(* IEC 61131-3 sources: neuroplc/results/scl_output (part 2) *)

      // MatMul 'l0_base': W + bias
      w2[0] := 0.6531532; w2[1] := 1.1509302; w2[2] := 0.8542801; w2[3] := 0.1212990; w2[4] := 0.6904182; w2[5] := -0.5414373; w2[6] := -0.9088417; w2[7] := -0.5722627;
      w2[8] := 0.8944874; w2[9] := 0.5538955; w2[10] := -1.0278374; w2[11] := -0.4903141; w2[12] := -0.1389806; w2[13] := 0.4674363; w2[14] := -1.0210936; w2[15] := -0.6274210;
      w2[16] := 0.2741612; w2[17] := 1.0625501; w2[18] := -0.9149109; w2[19] := -0.7328060; w2[20] := 0.7575151; w2[21] := -0.2042419; w2[22] := -0.2723309; w2[23] := -0.7191657;
      w2[24] := -0.0280776; w2[25] := 0.2011455; w2[26] := -0.3273573; w2[27] := -0.4418836; w2[28] := 1.2626092; w2[29] := 1.2265757; w2[30] := 1.5492810; w2[31] := -0.5662438;
      w2[32] := -0.9511591; w2[33] := 0.1725382; w2[34] := 1.2004387; w2[35] := -0.0104933; w2[36] := 1.5757133; w2[37] := 1.6623878; w2[38] := 1.2453479; w2[39] := 0.1729178;
      w2[40] := 0.2919613; w2[41] := 0.0309749; w2[42] := -0.6492561; w2[43] := -0.3796145; w2[44] := -0.5120577; w2[45] := 0.3172240; w2[46] := -0.4038502; w2[47] := 0.5928957;
      w2[48] := -0.5418487; w2[49] := -0.5144768; w2[50] := -0.7627655; w2[51] := 0.8234128; w2[52] := -0.4605753; w2[53] := -0.7895154; w2[54] := 0.0910844; w2[55] := -0.6752480;
      w2[56] := 0.0697802; w2[57] := -0.4284368; w2[58] := 0.0479970; w2[59] := 0.0784096; w2[60] := -0.0238369; w2[61] := 0.0168181; w2[62] := -0.8319796; w2[63] := 0.1763645;
      w2[64] := 0.2104895; w2[65] := 0.8926834; w2[66] := 0.6908084; w2[67] := 0.4001502; w2[68] := -0.3938401; w2[69] := 0.1085153; w2[70] := -0.6449838; w2[71] := -0.7566856;
      w2[72] := -0.0827282; w2[73] := 0.4948159; w2[74] := -1.1559126; w2[75] := -0.5277553; w2[76] := 0.8248507; w2[77] := 0.1181727; w2[78] := 0.7966241; w2[79] := 0.2058670;
      w2[80] := -0.8326430; w2[81] := -0.1626337; w2[82] := -0.0323979; w2[83] := -0.2344580; w2[84] := -1.5619131; w2[85] := -1.4697499; w2[86] := -1.8048265; w2[87] := -0.8762984;
      w2[88] := -1.3497895; w2[89] := -0.8686097; w2[90] := -0.9026392; w2[91] := -0.7284883; w2[92] := -1.7362306; w2[93] := -0.0363061; w2[94] := 1.1192808; w2[95] := 0.8043320;
      w2[96] := -0.1950512; w2[97] := -0.3716736; w2[98] := -0.4853409; w2[99] := -0.5649784; w2[100] := -0.4172391; w2[101] := 0.6161152; w2[102] := -0.6759697; w2[103] := 0.0904574;
      w2[104] := 0.5806844; w2[105] := 0.6348718; w2[106] := 0.7333751; w2[107] := 0.6839716; w2[108] := -0.3869329; w2[109] := 0.5344537; w2[110] := 0.9650685; w2[111] := 0.0383124;
      w2[112] := -0.8913731; w2[113] := -0.3576556; w2[114] := -0.6536014; w2[115] := -0.0847967; w2[116] := -0.0349820; w2[117] := 0.5889089; w2[118] := -0.2677067; w2[119] := -0.2245978;
      w2[120] := -0.5749647; w2[121] := -0.9168990; w2[122] := -0.6333076; w2[123] := -0.4074411; w2[124] := 0.4441338; w2[125] := 0.1501607; w2[126] := -0.1995225; w2[127] := 0.7596117;
      w2[128] := 0.0808029; w2[129] := -0.3484810; w2[130] := -0.0210259; w2[131] := 0.9137757; w2[132] := -0.7801852; w2[133] := -0.2238004; w2[134] := -0.3275166; w2[135] := -0.0392269;
      w2[136] := -0.2500529; w2[137] := 0.1511434; w2[138] := -0.2167200; w2[139] := 0.2951781; w2[140] := 0.3186197; w2[141] := 0.0769461; w2[142] := 0.4348049; w2[143] := -0.2419707;
      w2[144] := -0.3043656; w2[145] := -0.3270995; w2[146] := 0.5164679; w2[147] := 0.4538959; w2[148] := 0.2316195; w2[149] := 0.8929619; w2[150] := 1.3953813; w2[151] := 0.6482492;
      w2[152] := -0.2139386; w2[153] := -0.0555586; w2[154] := -0.2996079; w2[155] := -0.7336348; w2[156] := -0.7894226; w2[157] := 0.6769296; w2[158] := -1.0865229; w2[159] := 0.9084685;
      w2[160] := 0.4970312; w2[161] := 0.3730805; w2[162] := 0.6737831; w2[163] := 0.5160832; w2[164] := -0.8191277; w2[165] := 0.0919100; w2[166] := 0.4878978; w2[167] := -0.4577431;
      w2[168] := 0.5415249; w2[169] := 0.0459770; w2[170] := 0.2380498; w2[171] := 0.3544105; w2[172] := 0.0758338; w2[173] := 0.5700713; w2[174] := -0.3280728; w2[175] := 0.0073880;
      w2[176] := 0.9576581; w2[177] := -0.1927161; w2[178] := -0.5408630; w2[179] := 0.3759742; w2[180] := -0.3697540; w2[181] := -0.4095958; w2[182] := 0.2953050; w2[183] := -0.3224963;
      w2[184] := 0.4659955; w2[185] := 0.2666524; w2[186] := 0.7817978; w2[187] := -0.3882965; w2[188] := 0.5259117; w2[189] := 0.1157550; w2[190] := -0.0868794; w2[191] := 0.1442592;
      w2[192] := 0.4463586; w2[193] := -0.0788809; w2[194] := 0.3359323; w2[195] := 0.3131578; w2[196] := -0.2152938; w2[197] := 0.8472598; w2[198] := 0.6115276; w2[199] := -0.3911876;
      w2[200] := 0.0704370; w2[201] := -0.2515413; w2[202] := 0.8549601; w2[203] := 0.3596184; w2[204] := -0.5991781; w2[205] := -1.2437032; w2[206] := -0.1800027; w2[207] := -1.1388100;
      w2[208] := 0.5647227; w2[209] := 0.3254773; w2[210] := -0.8980638; w2[211] := 0.6457720; w2[212] := 0.9825901; w2[213] := -0.7528893; w2[214] := 0.0748151; w2[215] := 0.1365464;
      w2[216] := -0.6619212; w2[217] := -0.1892451; w2[218] := -0.3664528; w2[219] := -0.7725444; w2[220] := -0.1610090; w2[221] := -0.1782233; w2[222] := -0.1539104; w2[223] := -0.0613308;
      w2[224] := 1.0186411; w2[225] := -0.0857887; w2[226] := -0.3516517; w2[227] := 0.3065239; w2[228] := 0.0238268; w2[229] := 0.2399618; w2[230] := -0.2922754; w2[231] := -0.1875871;
      w2[232] := 1.1885412; w2[233] := -0.1608811; w2[234] := -1.1761448; w2[235] := -0.3997688; w2[236] := -1.0060421; w2[237] := 0.0516912; w2[238] := 0.4627137; w2[239] := -1.1369811;
      w2[240] := 0.6643242; w2[241] := 0.2780860; w2[242] := 0.0209994; w2[243] := -0.6893836; w2[244] := 0.5776726; w2[245] := -0.0303992; w2[246] := -0.2795104; w2[247] := -0.2218146;
      w2[248] := 0.4949092; w2[249] := 0.1933563; w2[250] := -0.3510525; w2[251] := 0.0224845; w2[252] := -1.5212339; w2[253] := -1.1815313; w2[254] := -1.4145346; w2[255] := 0.4340951;
      w2[256] := 0.3062091; w2[257] := 0.0455918; w2[258] := -0.3191082; w2[259] := 0.2872083; w2[260] := -1.7960831; w2[261] := -0.9681343; w2[262] := -0.2131347; w2[263] := -0.0914112;
      w2[264] := 0.4054331; w2[265] := -0.9982103; w2[266] := -0.5022178; w2[267] := 0.3359171; w2[268] := 0.8721167; w2[269] := -0.0940284; w2[270] := -1.9242376; w2[271] := 0.1256431;
      w2[272] := -0.4745836; w2[273] := 0.5358467; w2[274] := 0.1780284; w2[275] := -0.2262570; w2[276] := -0.6270480; w2[277] := -0.4930463; w2[278] := -0.6283804; w2[279] := 0.2633540;
      w2[280] := 0.2300479; w2[281] := 1.1844879; w2[282] := 0.6107946; w2[283] := -0.2428536; w2[284] := 0.4828842; w2[285] := 0.1695227; w2[286] := 0.5681323; w2[287] := 0.2884444;
      w2[288] := 0.2841129; w2[289] := -0.8758434; w2[290] := 0.2491129; w2[291] := -0.3859273; w2[292] := -0.4150312; w2[293] := 0.4644483; w2[294] := 0.1481924; w2[295] := -0.4265237;
      w2[296] := 0.3190451; w2[297] := -0.6888376; w2[298] := 0.8258311; w2[299] := 0.4234703; w2[300] := 0.0811714; w2[301] := -0.2619098; w2[302] := -1.0289083; w2[303] := -0.8263102;
      w2[304] := 0.5947338; w2[305] := -0.0104262; w2[306] := 0.4936709; w2[307] := 0.0368680; w2[308] := 0.0356015; w2[309] := 0.8885249; w2[310] := 0.5964210; w2[311] := -0.0492413;
      w2[312] := -0.1171272; w2[313] := -0.2020979; w2[314] := 0.5844330; w2[315] := -0.0603527; w2[316] := -0.1831383; w2[317] := -1.3109881; w2[318] := -0.5292199; w2[319] := 0.0204109;
      w2[320] := 0.2865884; w2[321] := -0.0319725; w2[322] := -0.1081036; w2[323] := 0.6079996; w2[324] := 0.7452201; w2[325] := -0.9360539; w2[326] := 0.2803982; w2[327] := 0.5940919;
      w2[328] := -0.3924443; w2[329] := -0.0010045; w2[330] := -0.2540028; w2[331] := -0.1956804; w2[332] := 0.3307257; w2[333] := -0.0851964; w2[334] := 0.0121359; w2[335] := 0.2464700;
      w2[336] := -1.3067886; w2[337] := -1.2725198; w2[338] := -1.4913075; w2[339] := 0.6236749; w2[340] := 0.3114894; w2[341] := 0.3706363; w2[342] := -0.5315891; w2[343] := 0.3905119;
      w2[344] := -1.4648223; w2[345] := -0.4327554; w2[346] := -0.1879684; w2[347] := -0.2010098; w2[348] := 0.5315167; w2[349] := -0.0843144; w2[350] := 0.0634309; w2[351] := 0.3992346;
      w2[352] := 0.3824810; w2[353] := -0.0483803; w2[354] := -0.2913157; w2[355] := 0.0982564; w2[356] := -0.4671767; w2[357] := 0.1136492; w2[358] := 0.0548117; w2[359] := -0.2728889;
      w2[360] := -0.4076180; w2[361] := -0.4225101; w2[362] := -0.2261286; w2[363] := 0.2782121; w2[364] := 0.7695327; w2[365] := 0.2566034; w2[366] := 0.1953621; w2[367] := 0.0408440;
      w2[368] := 0.0124786; w2[369] := 0.2488524; w2[370] := -0.5697264; w2[371] := 0.0825308; w2[372] := 0.8317476; w2[373] := -0.8402474; w2[374] := -1.0685767; w2[375] := -0.2165811;
      w2[376] := -0.4149429; w2[377] := -0.3753743; w2[378] := 0.1834853; w2[379] := 0.0865243; w2[380] := 0.7913322; w2[381] := -0.3387795; w2[382] := 0.5137359; w2[383] := -0.3165046;
      w2[384] := 0.2458227; w2[385] := 0.3609711; w2[386] := -0.3399727; w2[387] := -0.8827292; w2[388] := 0.4816631; w2[389] := 0.3397982; w2[390] := 0.1536530; w2[391] := 0.1695612;
      w2[392] := 0.5854009; w2[393] := -0.0813269; w2[394] := 0.1311246; w2[395] := 0.0674454; w2[396] := 0.2877986; w2[397] := -0.2290608; w2[398] := -0.6208226; w2[399] := -0.5486314;
      w2[400] := 0.9404889; w2[401] := 0.4580346; w2[402] := -0.5092251; w2[403] := -0.5765274; w2[404] := -0.4888373; w2[405] := 0.0444687; w2[406] := -0.2916232; w2[407] := -0.8206158;
      w2[408] := 0.2447187; w2[409] := 0.4721361; w2[410] := -0.6585346; w2[411] := -0.6879834; w2[412] := 0.5628800; w2[413] := 0.0532022; w2[414] := 0.1965619; w2[415] := 0.0561261;
      w2[416] := 0.2354458; w2[417] := 0.3610592; w2[418] := 0.0144084; w2[419] := 0.1184748; w2[420] := 0.0501975; w2[421] := 0.1787246; w2[422] := 0.4878071; w2[423] := 0.1703812;
      w2[424] := 0.1714815; w2[425] := -0.0600145; w2[426] := 0.7518312; w2[427] := 0.4750999; w2[428] := -0.1374112; w2[429] := 1.2641517; w2[430] := 1.2422327; w2[431] := 0.3578296;
      w2[432] := -0.3659381; w2[433] := 0.3438349; w2[434] := -0.3962274; w2[435] := -0.3011864; w2[436] := -0.1204108; w2[437] := 0.3932763; w2[438] := -0.0552154; w2[439] := 0.3200105;
      w2[440] := 0.7434683; w2[441] := 0.4552981; w2[442] := 0.4342712; w2[443] := 0.2647173; w2[444] := -0.2187249; w2[445] := -0.2678579; w2[446] := 0.1962206; w2[447] := -0.4789418;
      b3[0] := 0.0; b3[1] := 0.0; b3[2] := 0.0; b3[3] := 0.0; b3[4] := 0.0; b3[5] := 0.0; b3[6] := 0.0; b3[7] := 0.0;
      b3[8] := 0.0; b3[9] := 0.0; b3[10] := 0.0; b3[11] := 0.0; b3[12] := 0.0; b3[13] := 0.0; b3[14] := 0.0; b3[15] := 0.0;

      // BsplineLUT 'l1_bspline': grid + table
      g4[0] := -3.0000000; g4[1] := -2.5714286; g4[2] := -2.1428571; g4[3] := -1.7142857; g4[4] := -1.2857143; g4[5] := -0.8571429; g4[6] := -0.4285714; g4[7] := 0.0;
      g4[8] := 0.4285714; g4[9] := 0.8571429; g4[10] := 1.2857143; g4[11] := 1.7142857; g4[12] := 2.1428571; g4[13] := 2.5714286; g4[14] := 3.0000000;
      t5[0] := 0.1180185; t5[1] := 0.1203233; t5[2] := 0.1224589; t5[3] := 0.1244152; t5[4] := 0.1261825; t5[5] := 0.1277508; t5[6] := 0.1291103; t5[7] := 0.1302511;
      t5[8] := 0.1311632; t5[9] := 0.1318369; t5[10] := 0.1322627; t5[11] := 0.1324407; t5[12] := 0.1323814; t5[13] := 0.1320955; t5[14] := 0.1315938; t5[15] := 0.0842773;
      t5[16] := 0.0825064; t5[17] := 0.0806832; t5[18] := 0.0787976; t5[19] := 0.0768397; t5[20] := 0.0747991; t5[21] := 0.0726658; t5[22] := 0.0704296; t5[23] := 0.0680806;
      t5[24] := 0.0656084; t5[25] := 0.0630035; t5[26] := 0.0602665; t5[27] := 0.0574086; t5[28] := 0.0544416; t5[29] := 0.0513772; t5[30] := 0.0936770; t5[31] := 0.0899939;
      t5[32] := 0.0863021; t5[33] := 0.0826108; t5[34] := 0.0789293; t5[35] := 0.0752668; t5[36] := 0.0716325; t5[37] := 0.0680359; t5[38] := 0.0644860; t5[39] := 0.0609922;
      t5[40] := 0.0575636; t5[41] := 0.0542039; t5[42] := 0.0509117; t5[43] := 0.0476852; t5[44] := 0.0445227; t5[45] := 0.0226024; t5[46] := 0.0203358; t5[47] := 0.0180222;
      t5[48] := 0.0156702; t5[49] := 0.0132885; t5[50] := 0.0108859; t5[51] := 0.0084710; t5[52] := 0.0060526; t5[53] := 0.0036394; t5[54] := 0.0012401; t5[55] := -0.0011365;
      t5[56] := -0.0034818; t5[57] := -0.0057870; t5[58] := -0.0080435; t5[59] := -0.0102426; t5[60] := -0.0585543; t5[61] := -0.0502811; t5[62] := -0.0417866; t5[63] := -0.0330670;
      t5[64] := -0.0241186; t5[65] := -0.0149379; t5[66] := -0.0055211; t5[67] := 0.0041354; t5[68] := 0.0140353; t5[69] := 0.0241822; t5[70] := 0.0345793; t5[71] := 0.0452160;
      t5[72] := 0.0560676; t5[73] := 0.0671089; t5[74] := 0.0783146; t5[75] := 0.0506554; t5[76] := 0.0470260; t5[77] := 0.0433342; t5[78] := 0.0395754; t5[79] := 0.0357449;
      t5[80] := 0.0318381; t5[81] := 0.0278503; t5[82] := 0.0237768; t5[83] := 0.0196131; t5[84] := 0.0153543; t5[85] := 0.0109963; t5[86] := 0.0065434; t5[87] := 0.0020089;
      t5[88] := -0.0025934; t5[89] := -0.0072500; t5[90] := 0.0495298; t5[91] := 0.0382326; t5[92] := 0.0269749; t5[93] := 0.0157830; t5[94] := 0.0046829; t5[95] := -0.0062993;
      t5[96] := -0.0171372; t5[97] := -0.0278048; t5[98] := -0.0382758; t5[99] := -0.0485243; t5[100] := -0.0585243; t5[101] := -0.0682607; t5[102] := -0.0777291; t5[103] := -0.0869256;
      t5[104] := -0.0958461; t5[105] := 0.0110217; t5[106] := 0.0143777; t5[107] := 0.0176291; t5[108] := 0.0207730; t5[109] := 0.0238068; t5[110] := 0.0267275; t5[111] := 0.0295325;
      t5[112] := 0.0322190; t5[113] := 0.0347841; t5[114] := 0.0372252; t5[115] := 0.0395394; t5[116] := 0.0417255; t5[117] := 0.0437835; t5[118] := 0.0457136; t5[119] := 0.0475160;
      t5[120] := 0.1000672; t5[121] := 0.0975504; t5[122] := 0.0949741; t5[123] := 0.0923415; t5[124] := 0.0896557; t5[125] := 0.0869198; t5[126] := 0.0841368; t5[127] := 0.0813098;
      t5[128] := 0.0784420; t5[129] := 0.0755364; t5[130] := 0.0725962; t5[131] := 0.0696262; t5[132] := 0.0666327; t5[133] := 0.0636224; t5[134] := 0.0606016; t5[135] := -0.0637436;
      t5[136] := -0.0601492; t5[137] := -0.0563668; t5[138] := -0.0523824; t5[139] := -0.0481823; t5[140] := -0.0437526; t5[141] := -0.0390796; t5[142] := -0.0341494; t5[143] := -0.0289481;
      t5[144] := -0.0234621; t5[145] := -0.0176780; t5[146] := -0.0115977; t5[147] := -0.0052384; t5[148] := 0.0013820; t5[149] := 0.0082455; t5[150] := 0.0125032; t5[151] := 0.0077389;
      t5[152] := 0.0030834; t5[153] := -0.0014561; t5[154] := -0.0058727; t5[155] := -0.0101594; t5[156] := -0.0143091; t5[157] := -0.0183148; t5[158] := -0.0221695; t5[159] := -0.0258661;
      t5[160] := -0.0293979; t5[161] := -0.0327624; t5[162] := -0.0359621; t5[163] := -0.0389996; t5[164] := -0.0418773; t5[165] := 0.1193166; t5[166] := 0.1212150; t5[167] := 0.1228393;
      t5[168] := 0.1241749; t5[169] := 0.1252072; t5[170] := 0.1259215; t5[171] := 0.1263033; t5[172] := 0.1263380; t5[173] := 0.1260110; t5[174] := 0.1253076; t5[175] := 0.1242140;
      t5[176] := 0.1227300; t5[177] := 0.1208703; t5[178] := 0.1186500; t5[179] := 0.1160843; t5[180] := -0.1185704; t5[181] := -0.1148212; t5[182] := -0.1108735; t5[183] := -0.1067269;
      t5[184] := -0.1023809; t5[185] := -0.0978348; t5[186] := -0.0930883; t5[187] := -0.0881406; t5[188] := -0.0829914; t5[189] := -0.0776400; t5[190] := -0.0720863; t5[191] := -0.0663355;
      t5[192] := -0.0603990; t5[193] := -0.0542886; t5[194] := -0.0480157; t5[195] := 0.0583250; t5[196] := 0.0564782; t5[197] := 0.0548263; t5[198] := 0.0533813; t5[199] := 0.0521553;
      t5[200] := 0.0511605; t5[201] := 0.0504090; t5[202] := 0.0499130; t5[203] := 0.0496845; t5[204] := 0.0497356; t5[205] := 0.0500779; t5[206] := 0.0507077; t5[207] := 0.0516058;
      t5[208] := 0.0527522; t5[209] := 0.0541270; t5[210] := 0.1353638; t5[211] := 0.1313381; t5[212] := 0.1272324; t5[213] := 0.1230490; t5[214] := 0.1187897; t5[215] := 0.1144566;
      t5[216] := 0.1100518; t5[217] := 0.1055772; t5[218] := 0.1010349; t5[219] := 0.0964268; t5[220] := 0.0917550; t5[221] := 0.0870218; t5[222] := 0.0822297; t5[223] := 0.0773811;
      t5[224] := 0.0724786; t5[225] := -0.0180711; t5[226] := -0.0229253; t5[227] := -0.0277300; t5[228] := -0.0324813; t5[229] := -0.0371753; t5[230] := -0.0418079; t5[231] := -0.0463752;
      t5[232] := -0.0508733; t5[233] := -0.0552981; t5[234] := -0.0596458; t5[235] := -0.0639125; t5[236] := -0.0680959; t5[237] := -0.0721960; t5[238] := -0.0762126; t5[239] := -0.0801455;
      t5[240] := 0.1276658; t5[241] := 0.1281422; t5[242] := 0.1286489; t5[243] := 0.1291845; t5[244] := 0.1297478; t5[245] := 0.1303374; t5[246] := 0.1309519; t5[247] := 0.1315901;
      t5[248] := 0.1322506; t5[249] := 0.1329321; t5[250] := 0.1336332; t5[251] := 0.1343503; t5[252] := 0.1350780; t5[253] := 0.1358105; t5[254] := 0.1365422; t5[255] := 0.1341147;
      t5[256] := 0.1308563; t5[257] := 0.1273050; t5[258] := 0.1234552; t5[259] := 0.1193012; t5[260] := 0.1148372; t5[261] := 0.1100576; t5[262] := 0.1049567; t5[263] := 0.0995287;
      t5[264] := 0.0937679; t5[265] := 0.0876691; t5[266] := 0.0812383; t5[267] := 0.0744930; t5[268] := 0.0674512; t5[269] := 0.0601309; t5[270] := 0.0900934; t5[271] := 0.0884138;
      t5[272] := 0.0867445; t5[273] := 0.0850886; t5[274] := 0.0834493; t5[275] := 0.0818300; t5[276] := 0.0802338; t5[277] := 0.0786640; t5[278] := 0.0771239; t5[279] := 0.0756166;
      t5[280] := 0.0741453; t5[281] := 0.0727099; t5[282] := 0.0713072; t5[283] := 0.0699338; t5[284] := 0.0685862; t5[285] := 0.0413872; t5[286] := 0.0350636; t5[287] := 0.0287237;
      t5[288] := 0.0223717; t5[289] := 0.0160115; t5[290] := 0.0096474; t5[291] := 0.0032833; t5[292] := -0.0030765; t5[293] := -0.0094280; t5[294] := -0.0157671; t5[295] := -0.0220896;
      t5[296] := -0.0283901; t5[297] := -0.0346618; t5[298] := -0.0408980; t5[299] := -0.0470918; t5[300] := 0.0755875; t5[301] := 0.0739173; t5[302] := 0.0718717; t5[303] := 0.0694406;
      t5[304] := 0.0666140; t5[305] := 0.0633818; t5[306] := 0.0597340; t5[307] := 0.0556606; t5[308] := 0.0511514; t5[309] := 0.0461965; t5[310] := 0.0407865; t5[311] := 0.0349304;
      t5[312] := 0.0286561; t5[313] := 0.0219922; t5[314] := 0.0149673; t5[315] := 0.1297014; t5[316] := 0.1303879; t5[317] := 0.1309192; t5[318] := 0.1312868; t5[319] := 0.1314823;
      t5[320] := 0.1314970; t5[321] := 0.1313227; t5[322] := 0.1309508; t5[323] := 0.1303729; t5[324] := 0.1295806; t5[325] := 0.1285656; t5[326] := 0.1273265; t5[327] := 0.1258690;
      t5[328] := 0.1241989; t5[329] := 0.1223223; t5[330] := -0.0027479; t5[331] := 0.0012134; t5[332] := 0.0050790; t5[333] := 0.0088355; t5[334] := 0.0124699; t5[335] := 0.0159688;
      t5[336] := 0.0193190; t5[337] := 0.0225073; t5[338] := 0.0255204; t5[339] := 0.0283451; t5[340] := 0.0309686; t5[341] := 0.0333890; t5[342] := 0.0356160; t5[343] := 0.0376592;
      t5[344] := 0.0395288; t5[345] := 0.0290004; t5[346] := 0.0302992; t5[347] := 0.0316568; t5[348] := 0.0330863; t5[349] := 0.0346009; t5[350] := 0.0362138; t5[351] := 0.0379380;
      t5[352] := 0.0397869; t5[353] := 0.0417735; t5[354] := 0.0439110; t5[355] := 0.0462122; t5[356] := 0.0486769; t5[357] := 0.0512924; t5[358] := 0.0540451; t5[359] := 0.0569216;
      t5[360] := 0.0448184; t5[361] := 0.0512294; t5[362] := 0.0576943; t5[363] := 0.0642108; t5[364] := 0.0707761; t5[365] := 0.0773878; t5[366] := 0.0840433; t5[367] := 0.0907400;
      t5[368] := 0.0974754; t5[369] := 0.1042470; t5[370] := 0.1110519; t5[371] := 0.1178836; t5[372] := 0.1247314; t5[373] := 0.1315844; t5[374] := 0.1384318; t5[375] := 0.0079080;
      t5[376] := 0.0043265; t5[377] := 0.0007314; t5[378] := -0.0028650; t5[379] := -0.0064505; t5[380] := -0.0100129; t5[381] := -0.0135401; t5[382] := -0.0170198; t5[383] := -0.0204398;
      t5[384] := -0.0237880; t5[385] := -0.0270524; t5[386] := -0.0302289; t5[387] := -0.0333209; t5[388] := -0.0363325; t5[389] := -0.0392677; t5[390] := 0.1357616; t5[391] := 0.1397761;
      t5[392] := 0.1436628; t5[393] := 0.1474197; t5[394] := 0.1510451; t5[395] := 0.1545371; t5[396] := 0.1578940; t5[397] := 0.1611140; t5[398] := 0.1641951; t5[399] := 0.1671357;
      t5[400] := 0.1699338; t5[401] := 0.1725850; t5[402] := 0.1750826; t5[403] := 0.1774196; t5[404] := 0.1795891; t5[405] := 0.1128528; t5[406] := 0.1144198; t5[407] := 0.1158386;
      t5[408] := 0.1171095; t5[409] := 0.1182329; t5[410] := 0.1192093; t5[411] := 0.1200389; t5[412] := 0.1207222; t5[413] := 0.1212594; t5[414] := 0.1216511; t5[415] := 0.1218977;
      t5[416] := 0.1220020; t5[417] := 0.1219696; t5[418] := 0.1218062; t5[419] := 0.1215172; t5[420] := 0.1761363; t5[421] := 0.1778200; t5[422] := 0.1793493; t5[423] := 0.1807218;
      t5[424] := 0.1819351; t5[425] := 0.1829867; t5[426] := 0.1838742; t5[427] := 0.1845951; t5[428] := 0.1851470; t5[429] := 0.1855273; t5[430] := 0.1857340; t5[431] := 0.1857693;
      t5[432] := 0.1856408; t5[433] := 0.1853559; t5[434] := 0.1849222; t5[435] := -0.0491497; t5[436] := -0.0454618; t5[437] := -0.0415915; t5[438] := -0.0375284; t5[439] := -0.0332623;
      t5[440] := -0.0287830; t5[441] := -0.0240801; t5[442] := -0.0191433; t5[443] := -0.0139624; t5[444] := -0.0085271; t5[445] := -0.0028278; t5[446] := 0.0031299; t5[447] := 0.0093246;
      t5[448] := 0.0157340; t5[449] := 0.0223362; t5[450] := 0.1469728; t5[451] := 0.1491036; t5[452] := 0.1511741; t5[453] := 0.1531834; t5[454] := 0.1551309; t5[455] := 0.1570156;
      t5[456] := 0.1588368; t5[457] := 0.1605937; t5[458] := 0.1622854; t5[459] := 0.1639111; t5[460] := 0.1654701; t5[461] := 0.1669597; t5[462] := 0.1683763; t5[463] := 0.1697156;
      t5[464] := 0.1709738; t5[465] := 0.3216147; t5[466] := 0.3118152; t5[467] := 0.3017543; t5[468] := 0.2914528; t5[469] := 0.2809313; t5[470] := 0.2702106; t5[471] := 0.2593112;
      t5[472] := 0.2482539; t5[473] := 0.2370593; t5[474] := 0.2257481; t5[475] := 0.2143409; t5[476] := 0.2028543; t5[477] := 0.1913016; t5[478] := 0.1796954; t5[479] := 0.1680488;
      t5[480] := -0.0159183; t5[481] := -0.0107352; t5[482] := -0.0056755; t5[483] := -0.0007505; t5[484] := 0.0040286; t5[485] := 0.0086507; t5[486] := 0.0131043; t5[487] := 0.0173784;
      t5[488] := 0.0214616; t5[489] := 0.0253428; t5[490] := 0.0290110; t5[491] := 0.0324666; t5[492] := 0.0357209; t5[493] := 0.0387858; t5[494] := 0.0416731; t5[495] := -0.0254413;
      t5[496] := -0.0274388; t5[497] := -0.0293219; t5[498] := -0.0310746; t5[499] := -0.0326807; t5[500] := -0.0341243; t5[501] := -0.0353892; t5[502] := -0.0364594; t5[503] := -0.0373189;
      t5[504] := -0.0379516; t5[505] := -0.0383419; t5[506] := -0.0384855; t5[507] := -0.0383898; t5[508] := -0.0380625; t5[509] := -0.0375115; t5[510] := -0.0166281; t5[511] := -0.0149723;
      t5[512] := -0.0134576; t5[513] := -0.0120888; t5[514] := -0.0108707; t5[515] := -0.0098081; t5[516] := -0.0089057; t5[517] := -0.0081684; t5[518] := -0.0076009; t5[519] := -0.0072079;
      t5[520] := -0.0069941; t5[521] := -0.0069577; t5[522] := -0.0070906; t5[523] := -0.0073845; t5[524] := -0.0078309; t5[525] := -0.0174071; t5[526] := -0.0126844; t5[527] := -0.0078643;
      t5[528] := -0.0029462; t5[529] := 0.0020701; t5[530] := 0.0071853; t5[531] := 0.0123996; t5[532] := 0.0177135; t5[533] := 0.0231274; t5[534] := 0.0286418; t5[535] := 0.0342568;
      t5[536] := 0.0399670; t5[537] := 0.0457610; t5[538] := 0.0516272; t5[539] := 0.0575540; t5[540] := -0.0985392; t5[541] := -0.0994117; t5[542] := -0.1002845; t5[543] := -0.1011639;
      t5[544] := -0.1020565; t5[545] := -0.1029688; t5[546] := -0.1039072; t5[547] := -0.1048782; t5[548] := -0.1058883; t5[549] := -0.1069440; t5[550] := -0.1080513; t5[551] := -0.1092091;
      t5[552] := -0.1104083; t5[553] := -0.1116396; t5[554] := -0.1128937; t5[555] := 0.0001530; t5[556] := 0.0035909; t5[557] := 0.0070450; t5[558] := 0.0105171; t5[559] := 0.0140092;
      t5[560] := 0.0175231; t5[561] := 0.0210608; t5[562] := 0.0246240; t5[563] := 0.0282147; t5[564] := 0.0318347; t5[565] := 0.0354860; t5[566] := 0.0391708; t5[567] := 0.0428918;
      t5[568] := 0.0466516; t5[569] := 0.0504531; t5[570] := -0.0819526; t5[571] := -0.0816026; t5[572] := -0.0811294; t5[573] := -0.0805304; t5[574] := -0.0798034; t5[575] := -0.0789457;
      t5[576] := -0.0779550; t5[577] := -0.0768288; t5[578] := -0.0755645; t5[579] := -0.0741597; t5[580] := -0.0726123; t5[581] := -0.0709266; t5[582] := -0.0691139; t5[583] := -0.0671856;
      t5[584] := -0.0651534; t5[585] := 0.0965162; t5[586] := 0.0928315; t5[587] := 0.0891501; t5[588] := 0.0854817; t5[589] := 0.0818362; t5[590] := 0.0782233; t5[591] := 0.0746527;
      t5[592] := 0.0711343; t5[593] := 0.0676778; t5[594] := 0.0642930; t5[595] := 0.0609896; t5[596] := 0.0577725; t5[597] := 0.0546423; t5[598] := 0.0515992; t5[599] := 0.0486437;
      t5[600] := -0.2427283; t5[601] := -0.2398448; t5[602] := -0.2368635; t5[603] := -0.2337869; t5[604] := -0.2306173; t5[605] := -0.2273569; t5[606] := -0.2240082; t5[607] := -0.2205735;
      t5[608] := -0.2170550; t5[609] := -0.2134551; t5[610] := -0.2097761; t5[611] := -0.2060230; t5[612] := -0.2022031; t5[613] := -0.1983238; t5[614] := -0.1943926; t5[615] := -0.1351105;
      t5[616] := -0.1374491; t5[617] := -0.1394984; t5[618] := -0.1412510; t5[619] := -0.1426992; t5[620] := -0.1438354; t5[621] := -0.1446521; t5[622] := -0.1451416; t5[623] := -0.1452964;
      t5[624] := -0.1451089; t5[625] := -0.1445720; t5[626] := -0.1436916; t5[627] := -0.1424869; t5[628] := -0.1409778; t5[629] := -0.1391840; t5[630] := -0.0198544; t5[631] := -0.0241394;
      t5[632] := -0.0282630; t5[633] := -0.0322126; t5[634] := -0.0359753; t5[635] := -0.0395385; t5[636] := -0.0428895; t5[637] := -0.0460155; t5[638] := -0.0489037; t5[639] := -0.0515415;
      t5[640] := -0.0539166; t5[641] := -0.0560280; t5[642] := -0.0578859; t5[643] := -0.0595013; t5[644] := -0.0608852; t5[645] := 0.1033334; t5[646] := 0.0997555; t5[647] := 0.0962746;
      t5[648] := 0.0929015; t5[649] := 0.0896467; t5[650] := 0.0865207; t5[651] := 0.0835341; t5[652] := 0.0806975; t5[653] := 0.0780214; t5[654] := 0.0755164; t5[655] := 0.0731926;
      t5[656] := 0.0710490; t5[657] := 0.0690733; t5[658] := 0.0672527; t5[659] := 0.0655744; t5[660] := -0.0997362; t5[661] := -0.1019782; t5[662] := -0.1039813; t5[663] := -0.1057214;
      t5[664] := -0.1071745; t5[665] := -0.1083168; t5[666] := -0.1091242; t5[667] := -0.1095728; t5[668] := -0.1096387; t5[669] := -0.1092978; t5[670] := -0.1085273; t5[671] := -0.1073275;
      t5[672] := -0.1057235; t5[673] := -0.1037410; t5[674] := -0.1014061; t5[675] := -0.0270366; t5[676] := -0.0233783; t5[677] := -0.0198873; t5[678] := -0.0165889; t5[679] := -0.0135084;
      t5[680] := -0.0106710; t5[681] := -0.0081018; t5[682] := -0.0058263; t5[683] := -0.0038695; t5[684] := -0.0022567; t5[685] := -0.0010125; t5[686] := -0.0001434; t5[687] := 0.0003625;
      t5[688] := 0.0005178; t5[689] := 0.0003354; t5[690] := -0.0572062; t5[691] := -0.0531361; t5[692] := -0.0493332; t5[693] := -0.0458104; t5[694] := -0.0425804; t5[695] := -0.0396559;
      t5[696] := -0.0370498; t5[697] := -0.0347749; t5[698] := -0.0328439; t5[699] := -0.0312696; t5[700] := -0.0300643; t5[701] := -0.0292248; t5[702] := -0.0287326; t5[703] := -0.0285681;
      t5[704] := -0.0287122; t5[705] := 0.0384271; t5[706] := 0.0400259; t5[707] := 0.0414649; t5[708] := 0.0427437; t5[709] := 0.0438614; t5[710] := 0.0448175; t5[711] := 0.0456113;
      t5[712] := 0.0462421; t5[713] := 0.0467093; t5[714] := 0.0470122; t5[715] := 0.0471505; t5[716] := 0.0471296; t5[717] := 0.0469615; t5[718] := 0.0466583; t5[719] := 0.0462322;
      t5[720] := 0.0717728; t5[721] := 0.0695893; t5[722] := 0.0672396; t5[723] := 0.0647269; t5[724] := 0.0620541; t5[725] := 0.0592243; t5[726] := 0.0562403; t5[727] := 0.0531053;
      t5[728] := 0.0498221; t5[729] := 0.0463938; t5[730] := 0.0428236; t5[731] := 0.0391184; t5[732] := 0.0352894; t5[733] := 0.0313478; t5[734] := 0.0273048; t5[735] := -0.0450516;
      t5[736] := -0.0419416; t5[737] := -0.0386771; t5[738] := -0.0352532; t5[739] := -0.0316651; t5[740] := -0.0279082; t5[741] := -0.0239776; t5[742] := -0.0198686; t5[743] := -0.0155764;
      t5[744] := -0.0110964; t5[745] := -0.0064241; t5[746] := -0.0015652; t5[747] := 0.0034640; t5[748] := 0.0086470; t5[749] := 0.0139673; t5[750] := -0.0612851; t5[751] := -0.0675632;
      t5[752] := -0.0737045; t5[753] := -0.0796916; t5[754] := -0.0855072; t5[755] := -0.0911338; t5[756] := -0.0965540; t5[757] := -0.1017504; t5[758] := -0.1067057; t5[759] := -0.1114025;
      t5[760] := -0.1158238; t5[761] := -0.1199621; t5[762] := -0.1238200; t5[763] := -0.1274002; t5[764] := -0.1307057; t5[765] := -0.2006412; t5[766] := -0.1943896; t5[767] := -0.1878903;
      t5[768] := -0.1811593; t5[769] := -0.1742131; t5[770] := -0.1670678; t5[771] := -0.1597397; t5[772] := -0.1522450; t5[773] := -0.1446002; t5[774] := -0.1368213; t5[775] := -0.1289246;
      t5[776] := -0.1209250; t5[777] := -0.1128360; t5[778] := -0.1046710; t5[779] := -0.0964436; t5[780] := -0.1101506; t5[781] := -0.1094286; t5[782] := -0.1087262; t5[783] := -0.1080474;
      t5[784] := -0.1073962; t5[785] := -0.1067766; t5[786] := -0.1061925; t5[787] := -0.1056480; t5[788] := -0.1051469; t5[789] := -0.1046933; t5[790] := -0.1042911; t5[791] := -0.1039389;
      t5[792] := -0.1036309; t5[793] := -0.1033608; t5[794] := -0.1031222; t5[795] := -0.0820308; t5[796] := -0.0763831; t5[797] := -0.0706635; t5[798] := -0.0648856; t5[799] := -0.0590631;
      t5[800] := -0.0532094; t5[801] := -0.0473381; t5[802] := -0.0414628; t5[803] := -0.0355971; t5[804] := -0.0297545; t5[805] := -0.0239484; t5[806] := -0.0181894; t5[807] := -0.0124847;
      t5[808] := -0.0068417; t5[809] := -0.0012675; t5[810] := 0.0917091; t5[811] := 0.0912821; t5[812] := 0.0905308; t5[813] := 0.0894406; t5[814] := 0.0879973; t5[815] := 0.0861863;
      t5[816] := 0.0839933; t5[817] := 0.0814040; t5[818] := 0.0784038; t5[819] := 0.0749785; t5[820] := 0.0711144; t5[821] := 0.0668170; t5[822] := 0.0621115; t5[823] := 0.0570237;
      t5[824] := 0.0515798; t5[825] := -0.1294626; t5[826] := -0.1272798; t5[827] := -0.1249988; t5[828] := -0.1226242; t5[829] := -0.1201607; t5[830] := -0.1176130; t5[831] := -0.1149858;
      t5[832] := -0.1122837; t5[833] := -0.1095114; t5[834] := -0.1066737; t5[835] := -0.1037752; t5[836] := -0.1008182; t5[837] := -0.0978032; t5[838] := -0.0947306; t5[839] := -0.0916005;
      t5[840] := 0.0030728; t5[841] := 0.0004540; t5[842] := -0.0022056; t5[843] := -0.0048990; t5[844] := -0.0076197; t5[845] := -0.0103606; t5[846] := -0.0131151; t5[847] := -0.0158763;
      t5[848] := -0.0186375; t5[849] := -0.0213918; t5[850] := -0.0241325; t5[851] := -0.0268558; t5[852] := -0.0295605; t5[853] := -0.0322458; t5[854] := -0.0349107; t5[855] := -0.0715038;
      t5[856] := -0.0802228; t5[857] := -0.0888249; t5[858] := -0.0972798; t5[859] := -0.1055570; t5[860] := -0.1136262; t5[861] := -0.1214571; t5[862] := -0.1290192; t5[863] := -0.1362821;
      t5[864] := -0.1432156; t5[865] := -0.1497899; t5[866] := -0.1559936; t5[867] := -0.1618334; t5[868] := -0.1673172; t5[869] := -0.1724528; t5[870] := -0.0293459; t5[871] := -0.0276742;
      t5[872] := -0.0259024; t5[873] := -0.0240231; t5[874] := -0.0220287; t5[875] := -0.0199119; t5[876] := -0.0176651; t5[877] := -0.0152810; t5[878] := -0.0127520; t5[879] := -0.0100708;
      t5[880] := -0.0072302; t5[881] := -0.0042324; t5[882] := -0.0010891; t5[883] := 0.0021876; t5[884] := 0.0055856; t5[885] := -0.0198894; t5[886] := -0.0164613; t5[887] := -0.0130398;
      t5[888] := -0.0096217; t5[889] := -0.0062041; t5[890] := -0.0027840; t5[891] := 0.0006417; t5[892] := 0.0040759; t5[893] := 0.0075217; t5[894] := 0.0109821; t5[895] := 0.0144599;
      t5[896] := 0.0179544; t5[897] := 0.0214613; t5[898] := 0.0249760; t5[899] := 0.0284940; t5[900] := -0.0632152; t5[901] := -0.0687483; t5[902] := -0.0741381; t5[903] := -0.0793737;
      t5[904] := -0.0844447; t5[905] := -0.0893403; t5[906] := -0.0940500; t5[907] := -0.0985630; t5[908] := -0.1028687; t5[909] := -0.1069565; t5[910] := -0.1108161; t5[911] := -0.1144450;
      t5[912] := -0.1178493; t5[913] := -0.1210351; t5[914] := -0.1240087; t5[915] := 0.1738959; t5[916] := 0.1710729; t5[917] := 0.1680760; t5[918] := 0.1649032; t5[919] := 0.1615524;
      t5[920] := 0.1580214; t5[921] := 0.1543082; t5[922] := 0.1504108; t5[923] := 0.1463269; t5[924] := 0.1420544; t5[925] := 0.1375917; t5[926] := 0.1329436; t5[927] := 0.1281220;
      t5[928] := 0.1231391; t5[929] := 0.1180071; t5[930] := -0.0365145; t5[931] := -0.0358539; t5[932] := -0.0351557; t5[933] := -0.0344178; t5[934] := -0.0336381; t5[935] := -0.0328145;
      t5[936] := -0.0319450; t5[937] := -0.0310275; t5[938] := -0.0300599; t5[939] := -0.0290402; t5[940] := -0.0279663; t5[941] := -0.0268400; t5[942] := -0.0256666; t5[943] := -0.0244514;
      t5[944] := -0.0232000; t5[945] := -0.0122952; t5[946] := -0.0037388; t5[947] := 0.0045537; t5[948] := 0.0125514; t5[949] := 0.0202236; t5[950] := 0.0275394; t5[951] := 0.0344680;
      t5[952] := 0.0409785; t5[953] := 0.0470402; t5[954] := 0.0526223; t5[955] := 0.0576949; t5[956] := 0.0622538; t5[957] := 0.0663209; t5[958] := 0.0699191; t5[959] := 0.0730716;

      // MatMul 'l1_base': W + bias
      w6[0] := 0.0431468; w6[1] := -0.7218783; w6[2] := -0.7664040; w6[3] := 0.0446040; w6[4] := 0.6287033; w6[5] := -0.2051307; w6[6] := -0.3788366; w6[7] := 0.4265812;
      w6[8] := -0.5566995; w6[9] := 0.4906082; w6[10] := -0.1110822; w6[11] := 0.1812111; w6[12] := 0.4454913; w6[13] := -0.3052935; w6[14] := -0.5214026; w6[15] := -0.7138628;
      w6[16] := 0.9783757; w6[17] := -1.8518010; w6[18] := -0.4568165; w6[19] := -1.1427149; w6[20] := -0.0874276; w6[21] := -0.7568773; w6[22] := 0.8611937; w6[23] := -0.0933256;
      w6[24] := 0.6472971; w6[25] := -1.0294341; w6[26] := 0.3256389; w6[27] := 0.2590011; w6[28] := -0.7163869; w6[29] := 0.5744135; w6[30] := 0.3259708; w6[31] := -0.5870056;
      w6[32] := 0.2935589; w6[33] := 0.9891618; w6[34] := 1.2448254; w6[35] := 0.7247065; w6[36] := -0.0131453; w6[37] := 0.8092904; w6[38] := 0.1742139; w6[39] := -0.9718143;
      w6[40] := 0.1236900; w6[41] := 0.7221795; w6[42] := -0.6175265; w6[43] := -1.0537282; w6[44] := 0.4511162; w6[45] := -0.5315267; w6[46] := 0.3452142; w6[47] := 0.2253288;
      w6[48] := -1.2039654; w6[49] := 1.2277515; w6[50] := -0.3759507; w6[51] := 0.7626216; w6[52] := -0.6206948; w6[53] := 0.7239274; w6[54] := 0.0452536; w6[55] := 0.7874691;
      w6[56] := -0.5805001; w6[57] := -0.4060238; w6[58] := 0.7050563; w6[59] := 0.3644256; w6[60] := -0.6624428; w6[61] := -0.3291764; w6[62] := -0.9541196; w6[63] := 0.6871611;
      b7[0] := 0.0; b7[1] := 0.0; b7[2] := 0.0; b7[3] := 0.0;

(* ---- kan_iec_inference.st ---- *)
// NeuroPLC ˇŞ Vendor-neutral IEC 61131-3 ST inference block
// Graph: kan | Parameters in global data, logic in FB.

FUNCTION_BLOCK NeuroPLC_Inference

VAR_INPUT
    features : ARRAY[0..27] OF REAL;  // 28-D feature vector
END_VAR

VAR_OUTPUT
    fault_class : INT;  // 0=Normal, 1=InnerRace, 2=Ball, 3=OuterRace
    confidence : REAL;  // max softmax probability
END_VAR

VAR
    // ©¤©¤ Inference temporaries ©¤©¤
        v1 : ARRAY[0..27] OF REAL;  // silu output
        v3 : ARRAY[0..447] OF REAL;  // BsplineLUT output (1D: o*28+i)
        v2 : ARRAY[0..15] OF REAL;  // matmul output
        v4 : ARRAY[0..15] OF REAL;  // add merge
        v5 : ARRAY[0..15] OF REAL;  // silu output
        v7 : ARRAY[0..63] OF REAL;  // BsplineLUT output (1D: o*16+i)
        v6 : ARRAY[0..3] OF REAL;  // matmul output
        v8 : ARRAY[0..3] OF REAL;  // add merge
        v9 : ARRAY[0..3] OF REAL;  // softmax output

    // ©¤©¤ Temporary variables ©¤©¤
    i, o, j, lo, hi, idx, base : INT;
    sum, max_val, t_val : REAL;
END_VAR

BEGIN
    // ¨T¨T¨T Inference forward pass ¨T¨T¨T

        // Input: features[0..27]

        // StandardAct: silu
        FOR i := 0 TO 27 DO
            // SiLU = x / (1 + exp(-x))
            v1[i] := features[i] / (1.0 + EXP(-features[i]));
        END_FOR;

        // BsplineLUT: l0_bspline (16x28, 15 pts)
        FOR i := 0 TO 27 DO
            // Linear scan: find largest grid[j] <= input[i]
            lo := 0;
            FOR j := 1 TO 13 DO
                IF features[i] >= g0[j] THEN
                    lo := j;
                END_IF;
            END_FOR;
            hi := lo + 1;
            t_val := (features[i] - g0[lo]) /
                      (g0[hi] - g0[lo] + 1.0E-10);
            FOR o := 0 TO 15 DO
                base := (o * 28 + i) * 15;
                idx := o * 28 + i;
                v3[idx] :=
                    t1[base + lo] * (1.0 - t_val) +
                    t1[base + hi] * t_val;
            END_FOR;
        END_FOR;

        // MatMul: l0_base
        v2[0] := b3[0] + w2[0] * v1[0] + w2[1] * v1[1] + w2[2] * v1[2] + w2[3] * v1[3] + w2[4] * v1[4] + w2[5] * v1[5] + w2[6] * v1[6] + w2[7] * v1[7] + w2[8] * v1[8] + w2[9] * v1[9] + w2[10] * v1[10] + w2[11] * v1[11] + w2[12] * v1[12] + w2[13] * v1[13] + w2[14] * v1[14] + w2[15] * v1[15] + w2[16] * v1[16] + w2[17] * v1[17] + w2[18] * v1[18] + w2[19] * v1[19] + w2[20] * v1[20] + w2[21] * v1[21] + w2[22] * v1[22] + w2[23] * v1[23] + w2[24] * v1[24] + w2[25] * v1[25] + w2[26] * v1[26] + w2[27] * v1[27];
        v2[1] := b3[1] + w2[28] * v1[0] + w2[29] * v1[1] + w2[30] * v1[2] + w2[31] * v1[3] + w2[32] * v1[4] + w2[33] * v1[5] + w2[34] * v1[6] + w2[35] * v1[7] + w2[36] * v1[8] + w2[37] * v1[9] + w2[38] * v1[10] + w2[39] * v1[11] + w2[40] * v1[12] + w2[41] * v1[13] + w2[42] * v1[14] + w2[43] * v1[15] + w2[44] * v1[16] + w2[45] * v1[17] + w2[46] * v1[18] + w2[47] * v1[19] + w2[48] * v1[20] + w2[49] * v1[21] + w2[50] * v1[22] + w2[51] * v1[23] + w2[52] * v1[24] + w2[53] * v1[25] + w2[54] * v1[26] + w2[55] * v1[27];
        v2[2] := b3[2] + w2[56] * v1[0] + w2[57] * v1[1] + w2[58] * v1[2] + w2[59] * v1[3] + w2[60] * v1[4] + w2[61] * v1[5] + w2[62] * v1[6] + w2[63] * v1[7] + w2[64] * v1[8] + w2[65] * v1[9] + w2[66] * v1[10] + w2[67] * v1[11] + w2[68] * v1[12] + w2[69] * v1[13] + w2[70] * v1[14] + w2[71] * v1[15] + w2[72] * v1[16] + w2[73] * v1[17] + w2[74] * v1[18] + w2[75] * v1[19] + w2[76] * v1[20] + w2[77] * v1[21] + w2[78] * v1[22] + w2[79] * v1[23] + w2[80] * v1[24] + w2[81] * v1[25] + w2[82] * v1[26] + w2[83] * v1[27];
        v2[3] := b3[3] + w2[84] * v1[0] + w2[85] * v1[1] + w2[86] * v1[2] + w2[87] * v1[3] + w2[88] * v1[4] + w2[89] * v1[5] + w2[90] * v1[6] + w2[91] * v1[7] + w2[92] * v1[8] + w2[93] * v1[9] + w2[94] * v1[10] + w2[95] * v1[11] + w2[96] * v1[12] + w2[97] * v1[13] + w2[98] * v1[14] + w2[99] * v1[15] + w2[100] * v1[16] + w2[101] * v1[17] + w2[102] * v1[18] + w2[103] * v1[19] + w2[104] * v1[20] + w2[105] * v1[21] + w2[106] * v1[22] + w2[107] * v1[23] + w2[108] * v1[24] + w2[109] * v1[25] + w2[110] * v1[26] + w2[111] * v1[27];
        v2[4] := b3[4] + w2[112] * v1[0] + w2[113] * v1[1] + w2[114] * v1[2] + w2[115] * v1[3] + w2[116] * v1[4] + w2[117] * v1[5] + w2[118] * v1[6] + w2[119] * v1[7] + w2[120] * v1[8] + w2[121] * v1[9] + w2[122] * v1[10] + w2[123] * v1[11] + w2[124] * v1[12] + w2[125] * v1[13] + w2[126] * v1[14] + w2[127] * v1[15] + w2[128] * v1[16] + w2[129] * v1[17] + w2[130] * v1[18] + w2[131] * v1[19] + w2[132] * v1[20] + w2[133] * v1[21] + w2[134] * v1[22] + w2[135] * v1[23] + w2[136] * v1[24] + w2[137] * v1[25] + w2[138] * v1[26] + w2[139] * v1[27];
        v2[5] := b3[5] + w2[140] * v1[0] + w2[141] * v1[1] + w2[142] * v1[2] + w2[143] * v1[3] + w2[144] * v1[4] + w2[145] * v1[5] + w2[146] * v1[6] + w2[147] * v1[7] + w2[148] * v1[8] + w2[149] * v1[9] + w2[150] * v1[10] + w2[151] * v1[11] + w2[152] * v1[12] + w2[153] * v1[13] + w2[154] * v1[14] + w2[155] * v1[15] + w2[156] * v1[16] + w2[157] * v1[17] + w2[158] * v1[18] + w2[159] * v1[19] + w2[160] * v1[20] + w2[161] * v1[21] + w2[162] * v1[22] + w2[163] * v1[23] + w2[164] * v1[24] + w2[165] * v1[25] + w2[166] * v1[26] + w2[167] * v1[27];
        v2[6] := b3[6] + w2[168] * v1[0] + w2[169] * v1[1] + w2[170] * v1[2] + w2[171] * v1[3] + w2[172] * v1[4] + w2[173] * v1[5] + w2[174] * v1[6] + w2[175] * v1[7] + w2[176] * v1[8] + w2[177] * v1[9] + w2[178] * v1[10] + w2[179] * v1[11] + w2[180] * v1[12] + w2[181] * v1[13] + w2[182] * v1[14] + w2[183] * v1[15] + w2[184] * v1[16] + w2[185] * v1[17] + w2[186] * v1[18] + w2[187] * v1[19] + w2[188] * v1[20] + w2[189] * v1[21] + w2[190] * v1[22] + w2[191] * v1[23] + w2[192] * v1[24] + w2[193] * v1[25] + w2[194] * v1[26] + w2[195] * v1[27];
        v2[7] := b3[7] + w2[196] * v1[0] + w2[197] * v1[1] + w2[198] * v1[2] + w2[199] * v1[3] + w2[200] * v1[4] + w2[201] * v1[5] + w2[202] * v1[6] + w2[203] * v1[7] + w2[204] * v1[8] + w2[205] * v1[9] + w2[206] * v1[10] + w2[207] * v1[11] + w2[208] * v1[12] + w2[209] * v1[13] + w2[210] * v1[14] + w2[211] * v1[15] + w2[212] * v1[16] + w2[213] * v1[17] + w2[214] * v1[18] + w2[215] * v1[19] + w2[216] * v1[20] + w2[217] * v1[21] + w2[218] * v1[22] + w2[219] * v1[23] + w2[220] * v1[24] + w2[221] * v1[25] + w2[222] * v1[26] + w2[223] * v1[27];
        v2[8] := b3[8] + w2[224] * v1[0] + w2[225] * v1[1] + w2[226] * v1[2] + w2[227] * v1[3] + w2[228] * v1[4] + w2[229] * v1[5] + w2[230] * v1[6] + w2[231] * v1[7] + w2[232] * v1[8] + w2[233] * v1[9] + w2[234] * v1[10] + w2[235] * v1[11] + w2[236] * v1[12] + w2[237] * v1[13] + w2[238] * v1[14] + w2[239] * v1[15] + w2[240] * v1[16] + w2[241] * v1[17] + w2[242] * v1[18] + w2[243] * v1[19] + w2[244] * v1[20] + w2[245] * v1[21] + w2[246] * v1[22] + w2[247] * v1[23] + w2[248] * v1[24] + w2[249] * v1[25] + w2[250] * v1[26] + w2[251] * v1[27];
        v2[9] := b3[9] + w2[252] * v1[0] + w2[253] * v1[1] + w2[254] * v1[2] + w2[255] * v1[3] + w2[256] * v1[4] + w2[257] * v1[5] + w2[258] * v1[6] + w2[259] * v1[7] + w2[260] * v1[8] + w2[261] * v1[9] + w2[262] * v1[10] + w2[263] * v1[11] + w2[264] * v1[12] + w2[265] * v1[13] + w2[266] * v1[14] + w2[267] * v1[15] + w2[268] * v1[16] + w2[269] * v1[17] + w2[270] * v1[18] + w2[271] * v1[19] + w2[272] * v1[20] + w2[273] * v1[21] + w2[274] * v1[22] + w2[275] * v1[23] + w2[276] * v1[24] + w2[277] * v1[25] + w2[278] * v1[26] + w2[279] * v1[27];
        v2[10] := b3[10] + w2[280] * v1[0] + w2[281] * v1[1] + w2[282] * v1[2] + w2[283] * v1[3] + w2[284] * v1[4] + w2[285] * v1[5] + w2[286] * v1[6] + w2[287] * v1[7] + w2[288] * v1[8] + w2[289] * v1[9] + w2[290] * v1[10] + w2[291] * v1[11] + w2[292] * v1[12] + w2[293] * v1[13] + w2[294] * v1[14] + w2[295] * v1[15] + w2[296] * v1[16] + w2[297] * v1[17] + w2[298] * v1[18] + w2[299] * v1[19] + w2[300] * v1[20] + w2[301] * v1[21] + w2[302] * v1[22] + w2[303] * v1[23] + w2[304] * v1[24] + w2[305] * v1[25] + w2[306] * v1[26] + w2[307] * v1[27];
        v2[11] := b3[11] + w2[308] * v1[0] + w2[309] * v1[1] + w2[310] * v1[2] + w2[311] * v1[3] + w2[312] * v1[4] + w2[313] * v1[5] + w2[314] * v1[6] + w2[315] * v1[7] + w2[316] * v1[8] + w2[317] * v1[9] + w2[318] * v1[10] + w2[319] * v1[11] + w2[320] * v1[12] + w2[321] * v1[13] + w2[322] * v1[14] + w2[323] * v1[15] + w2[324] * v1[16] + w2[325] * v1[17] + w2[326] * v1[18] + w2[327] * v1[19] + w2[328] * v1[20] + w2[329] * v1[21] + w2[330] * v1[22] + w2[331] * v1[23] + w2[332] * v1[24] + w2[333] * v1[25] + w2[334] * v1[26] + w2[335] * v1[27];
        v2[12] := b3[12] + w2[336] * v1[0] + w2[337] * v1[1] + w2[338] * v1[2] + w2[339] * v1[3] + w2[340] * v1[4] + w2[341] * v1[5] + w2[342] * v1[6] + w2[343] * v1[7] + w2[344] * v1[8] + w2[345] * v1[9] + w2[346] * v1[10] + w2[347] * v1[11] + w2[348] * v1[12] + w2[349] * v1[13] + w2[350] * v1[14] + w2[351] * v1[15] + w2[352] * v1[16] + w2[353] * v1[17] + w2[354] * v1[18] + w2[355] * v1[19] + w2[356] * v1[20] + w2[357] * v1[21] + w2[358] * v1[22] + w2[359] * v1[23] + w2[360] * v1[24] + w2[361] * v1[25] + w2[362] * v1[26] + w2[363] * v1[27];
        v2[13] := b3[13] + w2[364] * v1[0] + w2[365] * v1[1] + w2[366] * v1[2] + w2[367] * v1[3] + w2[368] * v1[4] + w2[369] * v1[5] + w2[370] * v1[6] + w2[371] * v1[7] + w2[372] * v1[8] + w2[373] * v1[9] + w2[374] * v1[10] + w2[375] * v1[11] + w2[376] * v1[12] + w2[377] * v1[13] + w2[378] * v1[14] + w2[379] * v1[15] + w2[380] * v1[16] + w2[381] * v1[17] + w2[382] * v1[18] + w2[383] * v1[19] + w2[384] * v1[20] + w2[385] * v1[21] + w2[386] * v1[22] + w2[387] * v1[23] + w2[388] * v1[24] + w2[389] * v1[25] + w2[390] * v1[26] + w2[391] * v1[27];
        v2[14] := b3[14] + w2[392] * v1[0] + w2[393] * v1[1] + w2[394] * v1[2] + w2[395] * v1[3] + w2[396] * v1[4] + w2[397] * v1[5] + w2[398] * v1[6] + w2[399] * v1[7] + w2[400] * v1[8] + w2[401] * v1[9] + w2[402] * v1[10] + w2[403] * v1[11] + w2[404] * v1[12] + w2[405] * v1[13] + w2[406] * v1[14] + w2[407] * v1[15] + w2[408] * v1[16] + w2[409] * v1[17] + w2[410] * v1[18] + w2[411] * v1[19] + w2[412] * v1[20] + w2[413] * v1[21] + w2[414] * v1[22] + w2[415] * v1[23] + w2[416] * v1[24] + w2[417] * v1[25] + w2[418] * v1[26] + w2[419] * v1[27];
        v2[15] := b3[15] + w2[420] * v1[0] + w2[421] * v1[1] + w2[422] * v1[2] + w2[423] * v1[3] + w2[424] * v1[4] + w2[425] * v1[5] + w2[426] * v1[6] + w2[427] * v1[7] + w2[428] * v1[8] + w2[429] * v1[9] + w2[430] * v1[10] + w2[431] * v1[11] + w2[432] * v1[12] + w2[433] * v1[13] + w2[434] * v1[14] + w2[435] * v1[15] + w2[436] * v1[16] + w2[437] * v1[17] + w2[438] * v1[18] + w2[439] * v1[19] + w2[440] * v1[20] + w2[441] * v1[21] + w2[442] * v1[22] + w2[443] * v1[23] + w2[444] * v1[24] + w2[445] * v1[25] + w2[446] * v1[26] + w2[447] * v1[27];

        // Add: l0_merge
        FOR o := 0 TO 15 DO
            sum := v2[o];  // base path
            FOR i := 0 TO 27 DO
                idx := o * 28 + i;
                sum := sum + v3[idx];  // spline path (1D)
            END_FOR;
            v4[o] := sum;
        END_FOR;

        // StandardAct: silu
        FOR i := 0 TO 15 DO
            // SiLU = x / (1 + exp(-x))
            v5[i] := v4[i] / (1.0 + EXP(-v4[i]));
        END_FOR;

        // BsplineLUT: l1_bspline (4x16, 15 pts)
        FOR i := 0 TO 15 DO
            // Linear scan: find largest grid[j] <= input[i]
            lo := 0;
            FOR j := 1 TO 13 DO
                IF v4[i] >= g4[j] THEN
                    lo := j;
                END_IF;
            END_FOR;
            hi := lo + 1;
            t_val := (v4[i] - g4[lo]) /
                      (g4[hi] - g4[lo] + 1.0E-10);
            FOR o := 0 TO 3 DO
                base := (o * 16 + i) * 15;
                idx := o * 16 + i;
                v7[idx] :=
                    t5[base + lo] * (1.0 - t_val) +
                    t5[base + hi] * t_val;
            END_FOR;
        END_FOR;

        // MatMul: l1_base
        v6[0] := b7[0] + w6[0] * v5[0] + w6[1] * v5[1] + w6[2] * v5[2] + w6[3] * v5[3] + w6[4] * v5[4] + w6[5] * v5[5] + w6[6] * v5[6] + w6[7] * v5[7] + w6[8] * v5[8] + w6[9] * v5[9] + w6[10] * v5[10] + w6[11] * v5[11] + w6[12] * v5[12] + w6[13] * v5[13] + w6[14] * v5[14] + w6[15] * v5[15];
        v6[1] := b7[1] + w6[16] * v5[0] + w6[17] * v5[1] + w6[18] * v5[2] + w6[19] * v5[3] + w6[20] * v5[4] + w6[21] * v5[5] + w6[22] * v5[6] + w6[23] * v5[7] + w6[24] * v5[8] + w6[25] * v5[9] + w6[26] * v5[10] + w6[27] * v5[11] + w6[28] * v5[12] + w6[29] * v5[13] + w6[30] * v5[14] + w6[31] * v5[15];
        v6[2] := b7[2] + w6[32] * v5[0] + w6[33] * v5[1] + w6[34] * v5[2] + w6[35] * v5[3] + w6[36] * v5[4] + w6[37] * v5[5] + w6[38] * v5[6] + w6[39] * v5[7] + w6[40] * v5[8] + w6[41] * v5[9] + w6[42] * v5[10] + w6[43] * v5[11] + w6[44] * v5[12] + w6[45] * v5[13] + w6[46] * v5[14] + w6[47] * v5[15];
        v6[3] := b7[3] + w6[48] * v5[0] + w6[49] * v5[1] + w6[50] * v5[2] + w6[51] * v5[3] + w6[52] * v5[4] + w6[53] * v5[5] + w6[54] * v5[6] + w6[55] * v5[7] + w6[56] * v5[8] + w6[57] * v5[9] + w6[58] * v5[10] + w6[59] * v5[11] + w6[60] * v5[12] + w6[61] * v5[13] + w6[62] * v5[14] + w6[63] * v5[15];

        // Add: l1_merge
        FOR o := 0 TO 3 DO
            sum := v6[o];  // base path
            FOR i := 0 TO 15 DO
                idx := o * 16 + i;
                sum := sum + v7[idx];  // spline path (1D)
            END_FOR;
            v8[o] := sum;
        END_FOR;

        // Softmax
        max_val := v8[0];
        FOR i := 1 TO 3 DO
            IF v8[i] > max_val THEN
                max_val := v8[i];
            END_IF;
        END_FOR;
        sum := 0.0;
        FOR i := 0 TO 3 DO
            v9[i] := EXP(v8[i] - max_val);
            sum := sum + v9[i];
        END_FOR;
        FOR i := 0 TO 3 DO
            v9[i] := v9[i] / sum;
        END_FOR;

        // Argmax
        max_val := v9[0];
        fault_class := 0;
        FOR i := 1 TO 3 DO
            IF v9[i] > max_val THEN
                max_val := v9[i];
                fault_class := i;
            END_IF;
        END_FOR;
        confidence := max_val;

END_FUNCTION_BLOCK
